// TIA Portal V15.1 export
// export: Created 2020-06-12T07:35:55.9599609Z, ExportSetting None, DisplayName Totally Integrated Automation Portal, DisplayVersion V15.1, DisplayName TIA Portal Openness, DisplayVersion V15.1, DisplayName STEP 7 Professional, DisplayVersion V15.1, DisplayName STEP 7 Safety, DisplayVersion V15.1, DisplayName WinCC Advanced, DisplayVersion V15.1
FUNCTION "Fake_Output" : Void   // FC40, FBD
{ S7_Optimized_Access := 'TRUE' }
// stored: SetENOAutomatically False
   VAR_TEMP
      tClock : Bool;
   END_VAR
BEGIN

REGION Network 1: Check mechanics ES1LD1.EV01 +.EV02 (1)
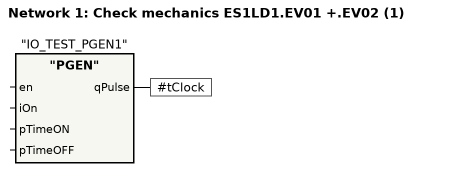
   "IO_TEST_PGEN1"(qPulse => #tClock);   // "PGEN"
END_REGION

REGION Network 2: Check mechanics ES1LD1.EV01 +.EV02 (2)
END_REGION
END_FUNCTION
